FUNCTION_BLOCK FB_Document
VAR_INPUT
END_VAR
VAR_OUTPUT
END_VAR
VAR
	_sContent		:STRING;
END_VAR

METHOD restoreFromMemento : BOOL
VAR_INPUT
	in_rstMemento		: REFERENCE TO ST_DocumentMemento;
END_VAR
IF NOT __ISVALIDREF(in_rstMemento) THEN
	RETURN;
END_IF

_sContent := in_rstMemento.sContent;

ADSLOGSTR(msgCtrlMask:= ADSLOG_MSGTYPE_ERROR, msgFmtStr:= 'Memento restored. Content: %s', strArg:= _sContent);
END_METHOD

PROPERTY sContent : String
GET
sContent := _sContent;
END_GET
END_PROPERTY

METHOD takeSnapshot : ST_DocumentMemento
takeSnapshot.sContent := _sContent;

ADSLOGSTR(msgCtrlMask:= ADSLOG_MSGTYPE_ERROR, msgFmtStr:= 'New Memento created. Content: %s', strArg:= _sContent);
END_METHOD

METHOD write : BOOL
VAR_INPUT
	in_sText	: STRING;
END_VAR
_sContent := in_sText;
END_METHOD

END_FUNCTION_BLOCK

(* stored: Version 1.1.0.1
   POU FB_Document: Id {a002d7e7-2009-46a9-835b-ea03020a0bd2}, SpecialFunc None
   Method restoreFromMemento: Id {ee5e9c02-17de-4aed-b37c-e875d6cdac20}
   Property sContent: Id {6f34124d-2ff2-4a3c-81d0-7e3cba3c31f6}
   Get Get: Id {a1b7c23d-4f3a-4c3d-a6c3-258edeb6f1b0}
   Method takeSnapshot: Id {fa9bde5e-34b4-47e1-be88-e62498a90cdc}
   Method write: Id {40621333-3db4-48f2-b4de-b4b51587dcc5} *)
